// Mitsubishi GX Works2 project: Start_Theo_Lan_Nhan   PLC: FX2N/FX2NC

PROGRAM MAIN
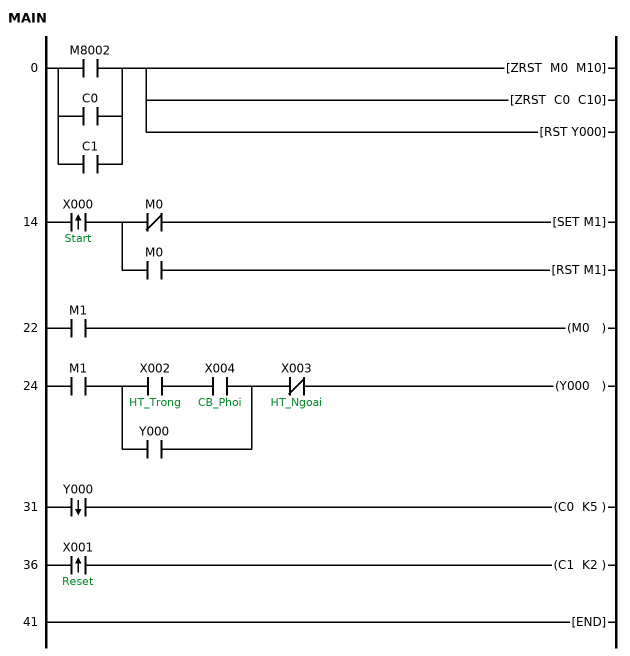
0     LD      M8002
      OR      C0
      OR      C1
      ZRST    M0 M10
      ZRST    C0 C10
      RST     Y000
14    LDP     X000  ; Start
      MPS
      ANI     M0
      SET     M1
      MPP
      AND     M0
      RST     M1
22    LD      M1
      OUT     M0
24    LD      M1
      LD      X002  ; HT_Trong
      AND     X004  ; CB_Phoi
      OR      Y000
      ANB
      ANI     X003  ; HT_Ngoai
      OUT     Y000
31    LDF     Y000
      OUT     C0 K5
36    LDP     X001  ; Reset
      OUT     C1 K2
41    END
END_PROGRAM
